// TwinCAT 3 PLC project Provider
// ProgramVersion: 3.1.4023.0
// libraries:
//   Tc2_Standard, * (Beckhoff Automation GmbH)
//   Tc2_System, * (Beckhoff Automation GmbH)
//   Tc3_JsonXml, * (Beckhoff Automation GmbH)
//   Tc3_Module, * (Beckhoff Automation GmbH)
//   Wordentec.Common, * (Wordentec Ltd)
//   Wordentec.Serial, * (Wordentec Ltd)
// project tree:
//   DUTs/ JsonDoc.TcDUT, ST_AnalogueValueWithBinaryStatus.TcDUT, ST_InputStatus.TcDUT, ST_IO_Status.TcDUT, ST_OutputStatus.TcDUT
//   GVLs/ API.TcGVL, IO.TcGVL
//   / PlcTask.TcTTO (not stored)
//   POUs/ FB_Math.TcPOU (not stored), MAIN.TcPOU (not stored), T_Data.TcPOU

// ---- DUTs/JsonDoc.TcDUT
TYPE
   JsonDoc : STRING(5000);
END_TYPE

// ---- DUTs/ST_AnalogueValueWithBinaryStatus.TcDUT
{attribute 'pack_mode' = '1'}
TYPE ST_AnalogueValueWithBinaryStatus :
STRUCT
	Value : REAL;
	BinaryStatus : BOOL;
END_STRUCT
END_TYPE

// ---- DUTs/ST_InputStatus.TcDUT
{attribute 'pack_mode' := '1'}
TYPE ST_InputStatus :
STRUCT
	T602_Platten_PSU : Wordentec_Serial.stTdkPsuStatus;
   T603_Source_PSU : Wordentec_Serial.stTdkPsuStatus;
   T606_Ch_1_Shutter_1_Open : BOOL;
   T606_Ch_2_Shutter_1_Closed : BOOL;
   T606_Ch_3_Bypass_Valve_Open : BOOL;
   T606_Ch_4_Bypass_Valve_Closed : BOOL;
   T607_Ch_1_Mains_OK : BOOL;
   T607_Ch_2_Spare : BOOL;
   T607_Ch_3_Spare : BOOL;
   T607_Ch_4_Spare : BOOL;
   T608_Ch_1_Shutter_1_Source_Baff : BOOL;
   T608_Ch_2_Shutter_2_Crystal : BOOL;
   T608_Ch_3_Purge_Valve : BOOL;
   T608_Ch_4_Bypass_Pump_Valve : BOOL;
   T614_Ch_1_Chamber_Water : ST_AnalogueValueWithBinaryStatus;
   T614_Ch_2_Water_In : ST_AnalogueValueWithBinaryStatus;
   T614_Ch_3_Water_Out : ST_AnalogueValueWithBinaryStatus;
   T614_Ch_4_Spare : ST_AnalogueValueWithBinaryStatus;
   T615_Ch_1_Platten_Temp : ST_AnalogueValueWithBinaryStatus;
   T615_Ch_2_Jig_Temperature : ST_AnalogueValueWithBinaryStatus;
   T615_Ch_3_spare : ST_AnalogueValueWithBinaryStatus;
   T615_Ch_4_spare : ST_AnalogueValueWithBinaryStatus;
   T616_Ch_1_Air_Pressure : ST_AnalogueValueWithBinaryStatus;
   T616_Ch_2_Water_Pressure : ST_AnalogueValueWithBinaryStatus;
   T617_Ch_1_Baratron_Pressure : ST_AnalogueValueWithBinaryStatus;
   T617_Ch_2_Nitorgen_Pressure : ST_AnalogueValueWithBinaryStatus;
	
END_STRUCT
END_TYPE

// ---- DUTs/ST_IO_Status.TcDUT
{attribute 'pack_mode' := '1'}
TYPE ST_IO_Status :
STRUCT
	inputs : ST_InputStatus;
	outputs : ST_OutputStatus;
END_STRUCT
END_TYPE

// ---- DUTs/ST_OutputStatus.TcDUT
{attribute 'pack_mode' := '1'}
TYPE ST_OutputStatus :
STRUCT
   T609_Ch_1_Platten_Heat_2K10 : Wordentec_Common.stDO_Status;
   T609_Ch_2_Platten_Cool_2K11 : Wordentec_Common.stDO_Status;
   T609_Ch_3_Source_1_2K12 : Wordentec_Common.stDO_Status;
   T609_Ch_4_Baratron_Isolation_Valve : Wordentec_Common.stDO_Status;
   T610_Ch_1_Is_Pumping_Light : Wordentec_Common.stDO_Status;
   T610_Ch_2_Has_a_fault_light : Wordentec_Common.stDO_Status;
   T610_Ch_3_Process_End_Light : Wordentec_Common.stDO_Status;
   T610_Ch_4_Is_Heating_Light : Wordentec_Common.stDO_Status;
	T611_Ch_1_Spare : Wordentec_Common.stDO_Status;
   T611_Ch_2_Spare : Wordentec_Common.stDO_Status;
   T611_Ch_3_Spare : Wordentec_Common.stDO_Status;
   T611_Ch_4_Spare : Wordentec_Common.stDO_Status;
   T612_Ch_1_Spare : Wordentec_Common.stDO_Status;
   T612_Ch_2_Spare : Wordentec_Common.stDO_Status;
   T613_Ch_1_Process_Rst_NO : Wordentec_Common.stDO_Status;
   T613_Ch_2_Process_Off_NC : Wordentec_Common.stDO_Status;
	T618_Ch_1_Spare : ST_AnalogueValueWithBinaryStatus;
   T618_Ch_2_Spare : ST_AnalogueValueWithBinaryStatus;
END_STRUCT
END_TYPE

// ---- GVLs/API.TcGVL
{attribute 'qualified_only'}
VAR_GLOBAL
	Data : T_Data;
END_VAR

// ---- GVLs/IO.TcGVL
{attribute 'qualified_only'}
VAR_GLOBAL
   IO_Status : ST_IO_Status;
END_VAR

// ---- POUs/T_Data.TcPOU
// provide API method calls to retreive IO status, Recipe Management Status and controller status.
FUNCTION_BLOCK T_Data
VAR_INPUT
END_VAR
VAR_OUTPUT
END_VAR
VAR
END_VAR

{attribute 'TcRpcEnable'}
METHOD PUBLIC GetIO : ST_IO_Status
VAR_INST
    cnt : INT;
END_VAR
GetIO := IO.IO_Status;
cnt := cnt + 1;
END_METHOD

{attribute 'TcRpcEnable'}
METHOD PUBLIC GetIOAsJson : JsonDoc
VAR_INST
    cnt : INT;
END_VAR
VAR 
	jsonDocToProp : FB_JsonReadWriteDatatype;
	sizeOfJDoc : UDINT;
END_VAR
VAR_INST
	sizeOfDoc : UDINT;
	jDoc : JsonDoc;
END_VAR
sizeOfDoc := SIZEOF(jDoc);
jsonDocToProp.GetJsonFromSymbol('ST_IO_Status',SIZEOF(IO.IO_Status), ADR(IO.IO_Status), sizeOfDoc, ADR(jDoc));
GetIOAsJson := jDoc;
cnt := cnt + 1;
END_METHOD

{attribute 'TcRpcEnable'}
METHOD PUBLIC SetIOAsJson : UDINT;
VAR_INPUT
	jDocIn : JsonDoc;
END_VAR
VAR_OUTPUT
	
END_VAR
VAR_INST
    cnt : INT;
END_VAR
VAR 
	jsonDocToProp : FB_JsonReadWriteDatatype;
	sizeOfJDoc : UDINT;
END_VAR
VAR_INST
	sizeOfDoc : UDINT;
	jDoc : JsonDoc;
	localIO : ST_IO_Status;
END_VAR
SetIOAsJson := SIZEOF(jDocIn);
jDoc := jDocIn;
jsonDocToProp.SetSymbolFromJson( jDocIn, 'ST_IO_Status',SIZEOF(localIo), ADR(localIo));
cnt := cnt + 1;
END_METHOD

END_FUNCTION_BLOCK
